FUNCTION_BLOCK ToFinalTreatment (* CAT Function Block Type *)
  (* Standard: 61499-2 *)
  (* Version 0.0, 6/21/2026, Schneider Electric, template *)
  PACKAGE SE.Nereda;
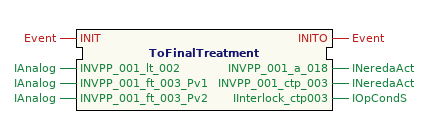
  EVENT_INPUT
    INIT;
  END_EVENT
  EVENT_OUTPUT
    INITO;
  END_EVENT
  SOCKETS
    INVPP_001_lt_002 : IAnalog;
    INVPP_001_ft_003_Pv1 : IAnalog;
  END_SOCKETS
  SOCKETS
    INVPP_001_ft_003_Pv2 : IAnalog; (* Process value (range considered) interface adapter *)
  END_SOCKETS
  PLUGS
    INVPP_001_a_018 : INeredaAct;
    INVPP_001_ctp_003 : INeredaAct;
  END_PLUGS
  PLUGS
    IInterlock_ctp003 : IOpCondS; (* Condition summary chain output to downstream block *)
  END_PLUGS
  (* 01 - FUNCTIONNAL INPUT INTERFACE *)
  (* 00 - INITIALIZATION *)
  (* 05 - LOGIC *)
  (* 06 - HMI INTERFACE *)
  (* 03 - FIELD INTERFACE *)
  (* 02 - FUNCTIONNAL OUTPUT INTERFACE *)
  (* Eflluent Pump ctp 003 & Valves 018 Control *)
  (* Interlock *)
  FBS
    IThis : ToFinalTreatment_HMI(QI := TRUE);
    NVPP_001_lt_002_Status : decodeStatus; {SET_ATTRIBUTE(Configuration.Component.HideUnusedPorts, )}
    NVPP_001_ft_003_Status : decodeStatus; {SET_ATTRIBUTE(Configuration.Component.HideUnusedPorts, )}
    PumpCmd : boolValueChanged;
    Valve18Cmd : boolValueChanged;
    PID_CTP_003 : PID; {SET_ATTRIBUTE(Configuration.Component.HideUnusedPorts, )}
    SpeedSpSmooth : RealValueChanged;
    ResetBtns : RESET_BTNs;
    PIDISc : PID_Manager;
    ControlLogic : TertFiltPumpMgr;
    StartLevelSpNotZero : COMPARE_1329C2AB45109BAAB(IN2 := 0.0); {SET_ATTRIBUTE(Configuration.GenericFBType.InterfaceParams, Runtime.Standard#CNT:=2;IN${CNT$}:REAL)} {SET_ATTRIBUTE(Configuration.Component.HideUnusedPorts, )}
    StopLevelSpNotZero : COMPARE_1329C2AB45109BAAB(IN2 := 0.0); {SET_ATTRIBUTE(Configuration.GenericFBType.InterfaceParams, Runtime.Standard#CNT:=2;IN${CNT$}:REAL)} {SET_ATTRIBUTE(Configuration.Component.HideUnusedPorts, )}
    StartLevelSp : COMPARE_1329C2AB45109BAAB; {SET_ATTRIBUTE(Configuration.GenericFBType.InterfaceParams, Runtime.Standard#CNT:=2;IN${CNT$}:REAL)} {SET_ATTRIBUTE(Configuration.Component.HideUnusedPorts, )}
    StopLevelSp : COMPARE_1329C2AB45109BAAB; {SET_ATTRIBUTE(Configuration.GenericFBType.InterfaceParams, Runtime.Standard#CNT:=2;IN${CNT$}:REAL)} {SET_ATTRIBUTE(Configuration.Component.HideUnusedPorts, )}
    StartCmd : AND_88A3DD8EC65DD11C; {SET_ATTRIBUTE(Configuration.GenericFBType.InterfaceParams, Runtime.Standard#CNT:=2;OUT:BOOL)}
    StopCmd : AND_88A3DD8EC65DD11C; {SET_ATTRIBUTE(Configuration.GenericFBType.InterfaceParams, Runtime.Standard#CNT:=2;OUT:BOOL)}
    DelayFlowAlarm : DelayedActive(pin_4E076A4928A0DFEF := TRUE, pin_1CE054BDD0AD4DEB := T#1m);
    LowLowFlow : AND_88A3DD8EC65DD11C; {SET_ATTRIBUTE(Configuration.GenericFBType.InterfaceParams, Runtime.Standard#CNT:=2;OUT:BOOL)}
    LowLowFlow_ctp003 : ilckCondItem(CondCause := Active1);
    PumpCtp003 : BOOL2INT;
    Valve18 : BOOL2INT;
    SpeedSp1 : SpeedSpFlowSensorFail;
  END_FBS
  EVENT_CONNECTIONS
    INVPP_001_lt_002.REQ_STATUS TO NVPP_001_lt_002_Status.REQ;
    INVPP_001_ft_003_Pv1.REQ_STATUS TO NVPP_001_ft_003_Status.REQ;
    StartCmd.CNF TO StopCmd.REQ;
    StartLevelSpNotZero.CNF TO StopLevelSpNotZero.REQ;
    StopLevelSpNotZero.CNF TO StartLevelSp.REQ;
    StartLevelSp.CNF TO StopLevelSp.REQ;
    StopLevelSp.CNF TO StartCmd.REQ;
    INVPP_001_lt_002.REQ TO StartLevelSpNotZero.REQ;
    LowLowFlow.CNF TO LowLowFlow_ctp003.REQ;
    INIT TO IThis.AABF4BC3AB55D4F4;
    IThis.6F082D2834F78A1D TO StartLevelSpNotZero.REQ;
    NVPP_001_ft_003_Status.CNF TO LowLowFlow.REQ;
    PIDISc.CE80458C9D5EF15A TO INITO;
    ControlLogic.STATE TO IThis.19BBDF43E4547D8F;
    ResetBtns.920962203CA54948 TO IThis.E7E377C8F1CEB610;
    PIDISc.CE80458C9D5EF15A TO IThis.8E2191486483827C;
    IThis.67A10949F5B1AAAB TO PIDISc.INIT;
    IThis.6F082D2834F78A1D TO PIDISc.REQ;
    IThis.63E33405E595E573 TO ControlLogic.REQ_ONOFF;
    IThis.B91C4BB13E300945 TO ResetBtns.AB695E9A35A20E19;
    IThis.B91C4BB13E300945 TO DelayFlowAlarm.C451626F7187F42D;
    StopCmd.CNF TO ControlLogic.REQ_LEVEL;
    INVPP_001_a_018.9CD053F8408797ED TO ControlLogic.FB_VALVE_018_STATE;
    INVPP_001_a_018.CC753684FA882790 TO ControlLogic.FB_VALVE_018_STATE;
    INVPP_001_ctp_003.9CD053F8408797ED TO ControlLogic.FB_PUMP_STATE;
    INVPP_001_ctp_003.CC753684FA882790 TO ControlLogic.FB_PUMP_STATE;
    ControlLogic.CNF_RUN_PUMP TO PumpCmd.REQ;
    ControlLogic.CNF_VALVE_a_018 TO Valve18Cmd.REQ;
    PumpCmd.CHD TO PumpCtp003.DD5870AA881150BB;
    Valve18Cmd.CHD TO Valve18.DD5870AA881150BB;
    PumpCtp003.6FC99A5BD1C38561 TO INVPP_001_ctp_003.0F1CDF9A9B4A227A;
    PumpCtp003.6FC99A5BD1C38561 TO PIDISc.REQ;
    Valve18.6FC99A5BD1C38561 TO INVPP_001_a_018.0F1CDF9A9B4A227A;
    PID_CTP_003.CNF TO SpeedSp1.B5D6B08FA2666F02;
    SpeedSpSmooth.93AE3729A9342678 TO INVPP_001_ctp_003.1E00729184986247;
    INVPP_001_ctp_003.9CD053F8408797ED TO DelayFlowAlarm.C451626F7187F42D;
    DelayFlowAlarm.DDA64CDC00519DA4 TO LowLowFlow.REQ;
    IThis.750F2719A617A972 TO ControlLogic.D0BF4D75F54A564B;
    IThis.750F2719A617A972 TO StartLevelSpNotZero.REQ;
    IThis.63E33405E595E573 TO StartLevelSpNotZero.REQ;
    SpeedSp1.1FEAADE7145F64BE TO SpeedSpSmooth.77F8F9CFF707DAFF;
    IThis.6F082D2834F78A1D TO SpeedSp1.B5D6B08FA2666F02;
    NVPP_001_ft_003_Status.CNF TO SpeedSp1.B5D6B08FA2666F02;
    INVPP_001_ft_003_Pv1.REQ TO SpeedSp1.B5D6B08FA2666F02;
  END_CONNECTIONS
  DATA_CONNECTIONS
    INVPP_001_lt_002.Status TO NVPP_001_lt_002_Status.Status;
    INVPP_001_ft_003_Pv1.Status TO NVPP_001_ft_003_Status.Status;
    INVPP_001_lt_002.Value TO StartLevelSp.IN1;
    INVPP_001_lt_002.Value TO StopLevelSp.IN1;
    StartLevelSpNotZero.NE TO StartCmd.IN1;
    StopLevelSpNotZero.NE TO StopCmd.IN1;
    StartLevelSp.GE TO StartCmd.IN2;
    StopLevelSp.LE TO StopCmd.IN2;
    LowLowFlow.OUT TO LowLowFlow_ctp003.CondSignal;
    IThis.D3B6E0932E654CC1 TO StartLevelSp.IN2;
    IThis.D3B6E0932E654CC1 TO StartLevelSpNotZero.IN1;
    IThis.06346DA38A4E8247 TO StopLevelSp.IN2;
    IThis.06346DA38A4E8247 TO StopLevelSpNotZero.IN1;
    NVPP_001_ft_003_Status.LoLoAlarm TO LowLowFlow.IN2;
    ControlLogic.State TO IThis.E29FE2D1F8D2DF4E;
    IThis.12A65F1451D1D9B3 TO PIDISc.Setpoint;
    IThis.4E9EAC06D5E10A12 TO ControlLogic.DB6583FA5935554F;
    IThis.FCF6192871811078 TO ControlLogic.OnOff;
    IThis.DC82B89A4AA2A4B1 TO ResetBtns.479D4538AEFD6EE1;
    IThis.DC82B89A4AA2A4B1 TO DelayFlowAlarm.45767490F5BA3A44;
    ControlLogic.RunPump TO PumpCmd.Input;
    ControlLogic.NVPP_001_a_018 TO Valve18Cmd.Input;
    StartCmd.OUT TO ControlLogic.HLevel;
    StopCmd.OUT TO ControlLogic.LLevel;
    INVPP_001_a_018.7F6CC7FEB9223DF3 TO ControlLogic.FbOpenValve018;
    INVPP_001_a_018.A8D6C4A1FDCCA991 TO ControlLogic.FbCloseValve018;
    INVPP_001_a_018.8A8A07EFCDA1443C TO ControlLogic.FbValve018Available;
    INVPP_001_ctp_003.B762734C094A7162 TO ControlLogic.FbPump;
    INVPP_001_ctp_003.D83B5BDEFA4D797C TO ControlLogic.71201958F060BBF6;
    INVPP_001_ctp_003.8A8A07EFCDA1443C TO ControlLogic.PumpNotAvailable;
    PumpCmd.Output TO PumpCtp003.4573FC8F228EB71D;
    Valve18Cmd.Output TO Valve18.4573FC8F228EB71D;
    PumpCtp003.A6DEF5F9C27C1848 TO INVPP_001_ctp_003.710D7FC54EE3F35A;
    Valve18.A6DEF5F9C27C1848 TO INVPP_001_a_018.710D7FC54EE3F35A;
    PumpCmd.Output TO PIDISc.RunPID;
    PID_CTP_003.Out TO SpeedSp1.4727B0C2E5DD09FB;
    SpeedSpSmooth.AA81B8787A42C5C8 TO INVPP_001_ctp_003.1BC103921BBFDA0B;
    INVPP_001_ctp_003.B762734C094A7162 TO DelayFlowAlarm.19546B227DE05AED;
    DelayFlowAlarm.614F3125208254F6 TO LowLowFlow.IN1;
    IThis.1D763E6DF1A35A69 TO ControlLogic.6A9F0F2DBB83FA68;
    SpeedSp1.87931CA83794BFFD TO SpeedSpSmooth.25B5287A5784F3EC;
    IThis.12A65F1451D1D9B3 TO SpeedSp1.3BE251DFC2E7905D;
    NVPP_001_ft_003_Status.FailAlarm TO SpeedSp1.1C28FEF37A13F67F;
    INVPP_001_ft_003_Pv1.ValueMax TO SpeedSp1.75C86D8B7647050C;
    INVPP_001_ft_003_Pv1.ValueMin TO SpeedSp1.B08827D02DBBFA97;
  END_CONNECTIONS
  ADAPTER_CONNECTIONS
    INVPP_001_ft_003_Pv2 TO PID_CTP_003.IPv;
    LowLowFlow_ctp003.ICondChainOut TO IInterlock_ctp003;
    PIDISc.FACD1DD4E791A86A TO PID_CTP_003.ISc;
  END_CONNECTIONS
END_FUNCTION_BLOCK
